TYPE ST_AutoAddsBoxes :
STRUCT
	Command	: ST_AutoAddsBoxesCommand;
	Status	: ST_AutoAddsBoxesStatus;
END_STRUCT
END_TYPE

(* stored: Version 1.1.0.1, ProductVersion 3.1.4024.13
   DUT ST_AutoAddsBoxes: Id {0483a49f-e72f-4da8-8385-6da5f9fca47b} *)
